FUNCTION Convert_WORD_TO_UINT : BOOL
VAR_INPUT
	in : WORD;
	out : REFERENCE TO UINT;
END_VAR
VAR
	converted : UINT;
END_VAR

converted := WORD_TO_UINT(in);

IF (UINT_TO_WORD(converted) <> in) THEN
	RETURN;
END_IF

out := converted;
Convert_WORD_TO_UINT := TRUE;

END_FUNCTION

(* stored: Version 1.1.0.1, ProductVersion 3.1.4024.12
   POU Convert_WORD_TO_UINT: Id {d82ee9ab-fc70-4718-a916-5aa6a8d81866}, SpecialFunc None *)
